// TIA Portal project "Assembler Control_Almaz" (V20)

(* hardware
DEVICE "S7-300/ET200M station_1"  S7-300 station
   slot 0: "Rail_0"  Rail  6ES7 390-1***0-0AA0
   slot 2: "PLC_1"  CPU 314C-2 PN/DP  6ES7 314-6EH04-0AB0  V3.3.18
      slot 2: "PROFINET interface_1"  PN-IO
         slot 1: "Port_1"  Port
         slot 2: "Port_2"  Port
      slot 5: "DI 24/DO 16_1"  DI24/DO16
      slot 6: "AI 5/AO 2_1"  AI5/AO2
      slot 7: "Count_1"  Counter
      slot 8: "Positioning_1"  Positioning
*)

// ===== PLC "PLC_1"  CPU 314C-2 PN/DP =====

VAR_GLOBAL   // PLC tag table "Output"
   "Move X" AT %Q0.0 : Bool;
   "Move Z" AT %Q0.1 : Bool;
   "Grab" AT %Q0.2 : Bool;
   "Lidsconveyor" AT %Q0.3 : Bool;
   "Clamp lid" AT %Q0.4 : Bool;
   "Pos. raise (lids)" AT %Q0.5 : Bool;
   "Bases conveyor" AT %Q0.6 : Bool;
   "Clamp base" AT %Q0.7 : Bool;
   "Pos. raise (bases)" AT %Q1.0 : Bool;
   "Start light" AT %Q1.1 : Bool;
   "Stop light" AT %Q1.2 : Bool;
   "Reset light" AT %Q1.3 : Bool;
   "Counter" AT %QD100 : DInt;
END_VAR

VAR_GLOBAL   // PLC tag table "Input"
   "Moving X" AT %I0.0 : Bool;
   "Moving Z" AT %I0.1 : Bool;
   "Item detected" AT %I0.2 : Bool;
   "Lid at place" AT %I0.3 : Bool;
   "Lid clamped" AT %I0.4 : Bool;
   "Pos. at limit (lids)" AT %I0.5 : Bool;
   "Base at place" AT %I0.6 : Bool;
   "Base clamped" AT %I0.7 : Bool;
   "Pos. at limit (bases)" AT %I1.0 : Bool;
   "Part leaving" AT %I1.1 : Bool;
   "Start" AT %I1.2 : Bool;
   "Reset" AT %I1.3 : Bool;
   "Stop" AT %I1.4 : Bool;
   "Emergency" AT %I1.5 : Bool;
   "Auto" AT %I1.6 : Bool;
   "Factory I/O Running" AT %I1.7 : Bool;
END_VAR

VAR_GLOBAL   // PLC tag table "Default tag table"
   "Tag_1" AT %M11.0 : Bool;
   "Base emitter" AT %Q1.4 : Bool;
   "Tag_2" AT %M11.3 : Bool;
   "Lids emitter" AT %Q1.5 : Bool;
   "Tag_3" AT %M11.1 : Bool;
   "Tag_4" AT %M20.1 : Bool;
   "Tag_5" AT %M0.0 : Bool;
   "Tag_6" AT %M2.6 : Bool;
   "Tag_7" AT %M0.1 : Bool;
   "Tag_8" AT %M0.2 : Bool;
   "Tag_9" AT %M12.3 : Bool;
   "Tag_10" AT %M0.3 : Bool;
   "Tag_11" AT %M0.4 : Bool;
   "Tag_12" AT %M2.0 : Bool;
   "Tag_13" AT %M0.6 : Bool;
   "Tag_14" AT %M1.5 : Bool;
   "Tag_15" AT %M1.2 : Bool;
   "Tag_16" AT %M2.2 : Bool;
   "Tag_17" AT %M50.3 : Bool;
   "Tag_18" AT %QD0 : DWord;
   "Tag_19" AT %MD0 : DWord;
   "Tag_20" AT %M10.0 : Bool;
   "Tag_21" AT %M50.1 : Bool;
   "Tag_22" AT %M11.7 : Bool;
   "Tag_23" AT %M2.4 : Bool;
   "Tag_24" AT %M12.0 : Bool;
   "Tag_25" AT %M12.6 : Bool;
   "Tag_26" AT %M1.1 : Bool;
   "Tag_27" AT %M2.1 : Bool;
END_VAR

ORGANIZATION_BLOCK "Main"   // OB1, LAD
TITLE = "Main Program Sweep (Cycle)"
{ S7_Optimized_Access := 'FALSE' }
VERSION : 0.1
   VAR_TEMP
      OB1_EV_CLASS : Byte;   // Bits 0-3 = 1 (Coming event), Bits 4-7 = 1 (Event class 1)
      OB1_SCAN_1 : Byte;   // 1 (Cold restart scan 1 of OB 1), 3 (Scan 2-n of OB 1)
      OB1_PRIORITY : Byte;   // Priority of OB Execution
      OB1_OB_NUMBR : Byte;   // 1 (Organization block 1, OB1)
      OB1_RESERVED_1 : Byte;   // Reserved for system
      OB1_RESERVED_2 : Byte;   // Reserved for system
      OB1_PREV_CYCLE : Int;   // Cycle time of previous OB1 scan (milliseconds)
      OB1_MIN_CYCLE : Int;   // Minimum cycle time of OB1 (milliseconds)
      OB1_MAX_CYCLE : Int;   // Maximum cycle time of OB1 (milliseconds)
      OB1_DATE_TIME : Date_And_Time;   // Date and time OB1 started
   END_VAR
   VAR_TEMP   // added for the SCL form of the ladder/FBD networks
      _w1 : Bool;
      _w2 : Bool;
      _w3 : Bool;
   END_VAR
BEGIN

REGION Network 1
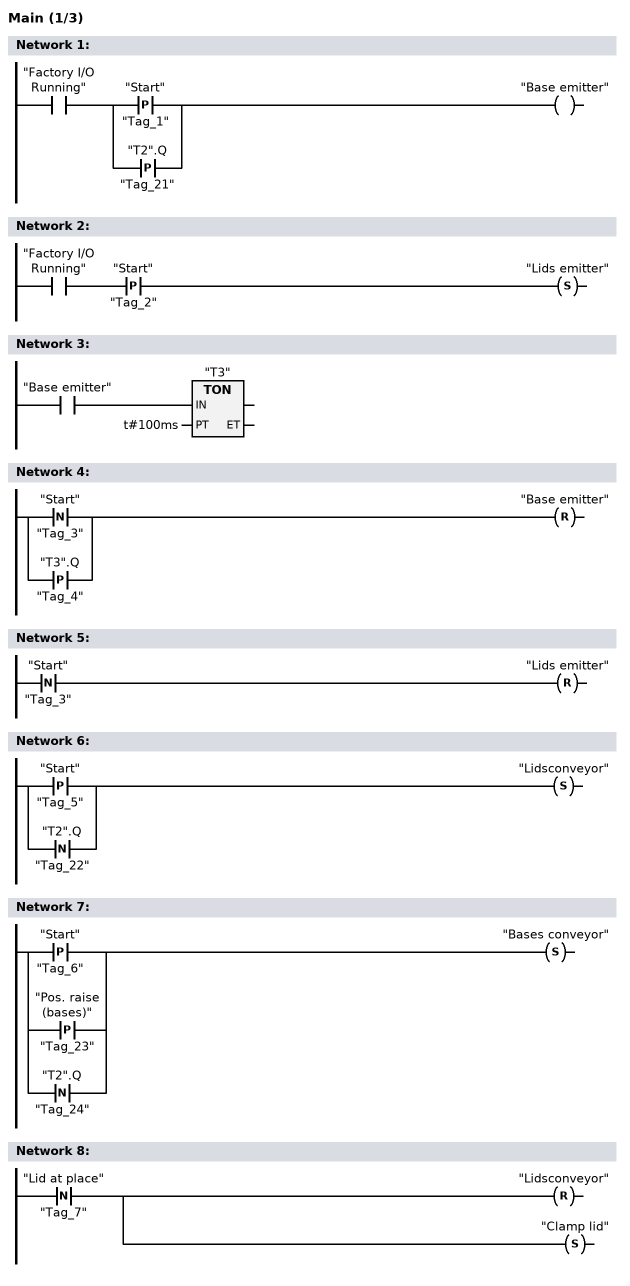
   RUNG wire#powerrail
      Contact( "Factory I/O Running" )
      wire#w1
      P_Contact(operand := "Start", bit := "Tag_1")
      wire#w2
      Coil( "Base emitter" )
   END_RUNG
   RUNG wire#w1
      P_Contact(operand := "T2".Q, bit := "Tag_21")
   END_RUNG wire#w2
   // the same network as SCL:
   #_w1 := "Factory I/O Running" AND "Start" AND NOT "Tag_1";   // rising edge of "Start"
   "Tag_1" := "Start";
   #_w2 := "Factory I/O Running" AND "T2".Q AND NOT "Tag_21";   // rising edge of "T2".Q
   "Tag_21" := "T2".Q;
   "Base emitter" := #_w1 OR #_w2;
END_REGION

REGION Network 2
   RUNG wire#powerrail
      Contact( "Factory I/O Running" )
      P_Contact(operand := "Start", bit := "Tag_2")
      S_Coil( "Lids emitter" )
   END_RUNG
   // the same network as SCL:
   #_w1 := "Factory I/O Running" AND "Start" AND NOT "Tag_2";   // rising edge of "Start"
   "Tag_2" := "Start";
   IF #_w1 THEN "Lids emitter" := TRUE; END_IF;
END_REGION

REGION Network 3
   "T3".TON(IN := "Base emitter", PT := t#100ms);
END_REGION

REGION Network 4
   RUNG wire#powerrail
      N_Contact(operand := "Start", bit := "Tag_3")
      wire#w1
      R_Coil( "Base emitter" )
   END_RUNG
   RUNG wire#powerrail
      P_Contact(operand := "T3".Q, bit := "Tag_4")
   END_RUNG wire#w1
   // the same network as SCL:
   #_w1 := NOT "Start" AND "Tag_3";   // falling edge of "Start"
   "Tag_3" := "Start";
   #_w2 := "T3".Q AND NOT "Tag_4";   // rising edge of "T3".Q
   "Tag_4" := "T3".Q;
   IF #_w1 OR #_w2 THEN "Base emitter" := FALSE; END_IF;
END_REGION

REGION Network 5
   RUNG wire#powerrail
      N_Contact(operand := "Start", bit := "Tag_3")
      R_Coil( "Lids emitter" )
   END_RUNG
   // the same network as SCL:
   #_w1 := NOT "Start" AND "Tag_3";   // falling edge of "Start"
   "Tag_3" := "Start";
   IF #_w1 THEN "Lids emitter" := FALSE; END_IF;
END_REGION

REGION Network 6
   RUNG wire#powerrail
      P_Contact(operand := "Start", bit := "Tag_5")
      wire#w1
      S_Coil( "Lidsconveyor" )
   END_RUNG
   RUNG wire#powerrail
      N_Contact(operand := "T2".Q, bit := "Tag_22")
   END_RUNG wire#w1
   // the same network as SCL:
   #_w1 := "Start" AND NOT "Tag_5";   // rising edge of "Start"
   "Tag_5" := "Start";
   #_w2 := NOT "T2".Q AND "Tag_22";   // falling edge of "T2".Q
   "Tag_22" := "T2".Q;
   IF #_w1 OR #_w2 THEN "Lidsconveyor" := TRUE; END_IF;
END_REGION

REGION Network 7
   RUNG wire#powerrail
      P_Contact(operand := "Start", bit := "Tag_6")
      wire#w1
      S_Coil( "Bases conveyor" )
   END_RUNG
   RUNG wire#powerrail
      P_Contact(operand := "Pos. raise (bases)", bit := "Tag_23")
   END_RUNG wire#w1
   RUNG wire#powerrail
      N_Contact(operand := "T2".Q, bit := "Tag_24")
   END_RUNG wire#w1
   // the same network as SCL:
   #_w1 := "Start" AND NOT "Tag_6";   // rising edge of "Start"
   "Tag_6" := "Start";
   #_w2 := "Pos. raise (bases)" AND NOT "Tag_23";   // rising edge of "Pos. raise (bases)"
   "Tag_23" := "Pos. raise (bases)";
   #_w3 := NOT "T2".Q AND "Tag_24";   // falling edge of "T2".Q
   "Tag_24" := "T2".Q;
   IF #_w1 OR #_w2 OR #_w3 THEN "Bases conveyor" := TRUE; END_IF;
END_REGION

REGION Network 8
   RUNG wire#powerrail
      N_Contact(operand := "Lid at place", bit := "Tag_7")
      wire#w1
      R_Coil( "Lidsconveyor" )
   END_RUNG
   RUNG wire#w1
      S_Coil( "Clamp lid" )
   END_RUNG
   // the same network as SCL:
   #_w1 := NOT "Lid at place" AND "Tag_7";   // falling edge of "Lid at place"
   "Tag_7" := "Lid at place";
   IF #_w1 THEN
       "Lidsconveyor" := FALSE;
       "Clamp lid" := TRUE;
   END_IF;
END_REGION

REGION Network 9
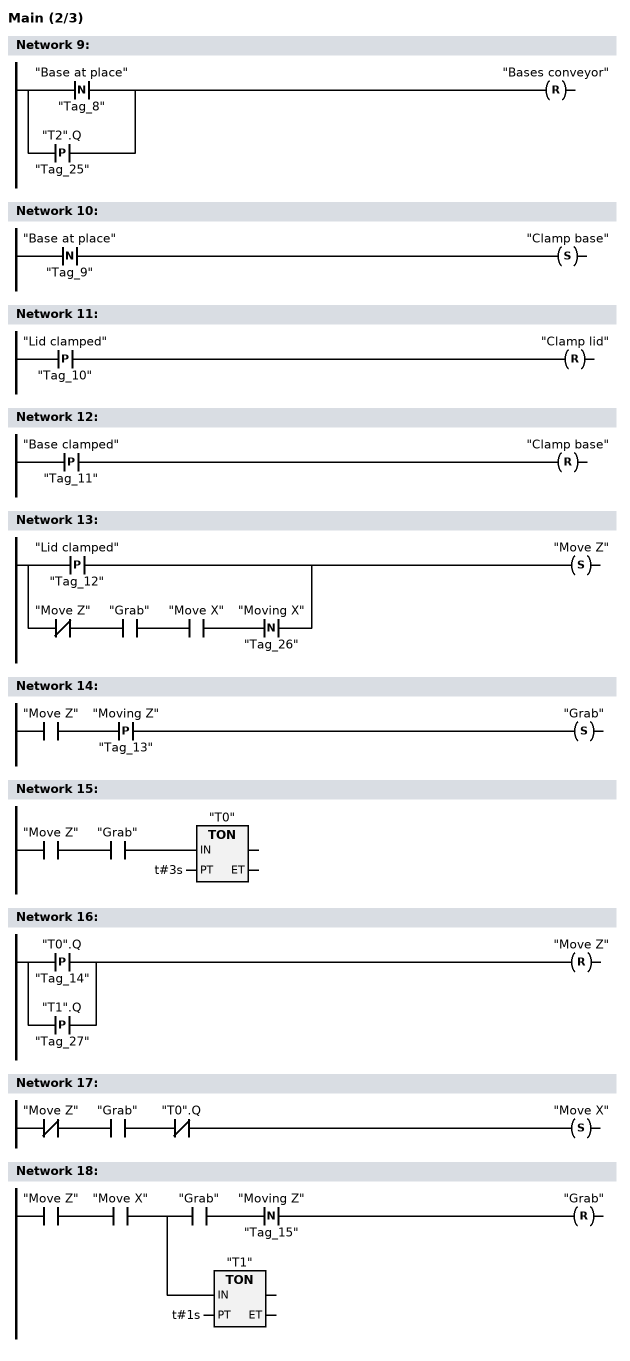
   RUNG wire#powerrail
      N_Contact(operand := "Base at place", bit := "Tag_8")
      wire#w1
      R_Coil( "Bases conveyor" )
   END_RUNG
   RUNG wire#powerrail
      P_Contact(operand := "T2".Q, bit := "Tag_25")
   END_RUNG wire#w1
   // the same network as SCL:
   #_w1 := NOT "Base at place" AND "Tag_8";   // falling edge of "Base at place"
   "Tag_8" := "Base at place";
   #_w2 := "T2".Q AND NOT "Tag_25";   // rising edge of "T2".Q
   "Tag_25" := "T2".Q;
   IF #_w1 OR #_w2 THEN "Bases conveyor" := FALSE; END_IF;
END_REGION

REGION Network 10
   RUNG wire#powerrail
      N_Contact(operand := "Base at place", bit := "Tag_9")
      S_Coil( "Clamp base" )
   END_RUNG
   // the same network as SCL:
   #_w1 := NOT "Base at place" AND "Tag_9";   // falling edge of "Base at place"
   "Tag_9" := "Base at place";
   IF #_w1 THEN "Clamp base" := TRUE; END_IF;
END_REGION

REGION Network 11
   RUNG wire#powerrail
      P_Contact(operand := "Lid clamped", bit := "Tag_10")
      R_Coil( "Clamp lid" )
   END_RUNG
   // the same network as SCL:
   #_w1 := "Lid clamped" AND NOT "Tag_10";   // rising edge of "Lid clamped"
   "Tag_10" := "Lid clamped";
   IF #_w1 THEN "Clamp lid" := FALSE; END_IF;
END_REGION

REGION Network 12
   RUNG wire#powerrail
      P_Contact(operand := "Base clamped", bit := "Tag_11")
      R_Coil( "Clamp base" )
   END_RUNG
   // the same network as SCL:
   #_w1 := "Base clamped" AND NOT "Tag_11";   // rising edge of "Base clamped"
   "Tag_11" := "Base clamped";
   IF #_w1 THEN "Clamp base" := FALSE; END_IF;
END_REGION

REGION Network 13
   RUNG wire#powerrail
      P_Contact(operand := "Lid clamped", bit := "Tag_12")
      wire#w1
      S_Coil( "Move Z" )
   END_RUNG
   RUNG wire#powerrail
      I_Contact( "Move Z" )
      Contact( "Grab" )
      Contact( "Move X" )
      N_Contact(operand := "Moving X", bit := "Tag_26")
   END_RUNG wire#w1
   // the same network as SCL:
   #_w1 := "Lid clamped" AND NOT "Tag_12";   // rising edge of "Lid clamped"
   "Tag_12" := "Lid clamped";
   #_w2 := NOT "Move Z" AND "Grab" AND "Move X" AND NOT "Moving X" AND "Tag_26";   // falling edge of "Moving X"
   "Tag_26" := "Moving X";
   IF #_w1 OR #_w2 THEN "Move Z" := TRUE; END_IF;
END_REGION

REGION Network 14
   RUNG wire#powerrail
      Contact( "Move Z" )
      P_Contact(operand := "Moving Z", bit := "Tag_13")
      S_Coil( "Grab" )
   END_RUNG
   // the same network as SCL:
   #_w1 := "Move Z" AND "Moving Z" AND NOT "Tag_13";   // rising edge of "Moving Z"
   "Tag_13" := "Moving Z";
   IF #_w1 THEN "Grab" := TRUE; END_IF;
END_REGION

REGION Network 15
   "T0".TON(IN := "Move Z" AND "Grab", PT := t#3s);
END_REGION

REGION Network 16
   RUNG wire#powerrail
      P_Contact(operand := "T0".Q, bit := "Tag_14")
      wire#w1
      R_Coil( "Move Z" )
   END_RUNG
   RUNG wire#powerrail
      P_Contact(operand := "T1".Q, bit := "Tag_27")
   END_RUNG wire#w1
   // the same network as SCL:
   #_w1 := "T0".Q AND NOT "Tag_14";   // rising edge of "T0".Q
   "Tag_14" := "T0".Q;
   #_w2 := "T1".Q AND NOT "Tag_27";   // rising edge of "T1".Q
   "Tag_27" := "T1".Q;
   IF #_w1 OR #_w2 THEN "Move Z" := FALSE; END_IF;
END_REGION

REGION Network 17
   RUNG wire#powerrail
      I_Contact( "Move Z" )
      Contact( "Grab" )
      I_Contact( "T0".Q )
      S_Coil( "Move X" )
   END_RUNG
   // the same network as SCL:
   IF NOT "Move Z" AND "Grab" AND NOT "T0".Q THEN "Move X" := TRUE; END_IF;
END_REGION

REGION Network 18
   #_w1 := "Move Z" AND "Move X";
   #_w2 := #_w1 AND "Grab" AND NOT "Moving Z" AND "Tag_15";   // falling edge of "Moving Z"
   "Tag_15" := "Moving Z";
   IF #_w2 THEN "Grab" := FALSE; END_IF;
   "T1".TON(IN := #_w1, PT := t#1s);
END_REGION

REGION Network 19
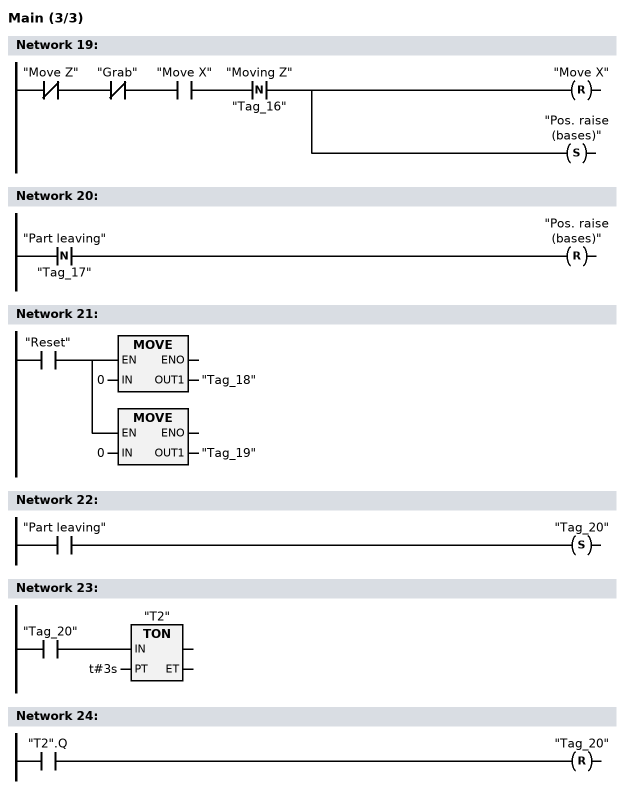
   RUNG wire#powerrail
      I_Contact( "Move Z" )
      I_Contact( "Grab" )
      Contact( "Move X" )
      N_Contact(operand := "Moving Z", bit := "Tag_16")
      wire#w1
      R_Coil( "Move X" )
   END_RUNG
   RUNG wire#w1
      S_Coil( "Pos. raise (bases)" )
   END_RUNG
   // the same network as SCL:
   #_w1 := NOT "Move Z" AND NOT "Grab" AND "Move X" AND NOT "Moving Z" AND "Tag_16";   // falling edge of "Moving Z"
   "Tag_16" := "Moving Z";
   IF #_w1 THEN
       "Move X" := FALSE;
       "Pos. raise (bases)" := TRUE;
   END_IF;
END_REGION

REGION Network 20
   RUNG wire#powerrail
      N_Contact(operand := "Part leaving", bit := "Tag_17")
      R_Coil( "Pos. raise (bases)" )
   END_RUNG
   // the same network as SCL:
   #_w1 := NOT "Part leaving" AND "Tag_17";   // falling edge of "Part leaving"
   "Tag_17" := "Part leaving";
   IF #_w1 THEN "Pos. raise (bases)" := FALSE; END_IF;
END_REGION

REGION Network 21
   RUNG wire#powerrail
      Contact( "Reset" )
      wire#w1
      { S7_GenerateENO := "TRUE" } Move(in := 0, out1 => "Tag_18")
   END_RUNG
   RUNG wire#w1
      { S7_GenerateENO := "TRUE" } Move(in := 0, out1 => "Tag_19")
   END_RUNG
   // the same network as SCL:
   IF "Reset" THEN
       "Tag_18" := 0;
       "Tag_19" := 0;
   END_IF;
END_REGION

REGION Network 22
   RUNG wire#powerrail
      Contact( "Part leaving" )
      S_Coil( "Tag_20" )
   END_RUNG
   // the same network as SCL:
   IF "Part leaving" THEN "Tag_20" := TRUE; END_IF;
END_REGION

REGION Network 23
   "T2".TON(IN := "Tag_20", PT := t#3s);
END_REGION

REGION Network 24
   RUNG wire#powerrail
      Contact( "T2".Q )
      R_Coil( "Tag_20" )
   END_RUNG
   // the same network as SCL:
   IF "T2".Q THEN "Tag_20" := FALSE; END_IF;
END_REGION
END_ORGANIZATION_BLOCK